SUBAPPLICATION Select_EnableOk (* Leitet aus 2 Bools (bEnable + bOk) einen von 3 Werten ab: valDisabled (bEnable=FALSE) / valOk (bEnable=TRUE, bOk=TRUE) / valFault (bEnable=TRUE, bOk=FALSE). Generischer 2-stufiger F_SEL - die 3 Werte sind Parameter, nicht auf Farben beschraenkt. *)
  (* Standard: 61499-2; Description: Copyright (c) 2026 Meisterschulen am Ostbahnhof This program and the accompanying materials are made available under the terms of the Eclipse Public License 2.0 which is available at https://www.eclipse.org/legal/epl-2.0/ SPDX-License-Identifier: EPL-2.0 *)
  (* Version 1.0, 2026-08-31, Franz Höpfinger, Meisterschulen am Ostbahnhof, Extrahiert aus Q_BackgroundColour_EnableOk - die reine 2-Bool-zu-1-von-3-Werten-Logik, entkoppelt von der VT-Hintergrundfarben-Anwendung *)
  PACKAGE MyLib::sys;
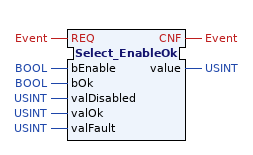
  EVENT_INPUT
    REQ; (* Neu auswerten - bEnable und bOk werden zusammen mitgegeben *)
  END_EVENT
  EVENT_OUTPUT
    CNF; (* Wert berechnet *)
  END_EVENT
  VAR_INPUT
    bEnable : BOOL; (* Aktiviert *)
    bOk : BOOL; (* OK-Zustand (nur relevant wenn bEnable=TRUE) *)
    valDisabled : USINT; (* Ausgabewert wenn bEnable=FALSE - einmalig bei Instanziierung per Parameter gesetzt *)
    valOk : USINT; (* Ausgabewert wenn bEnable=TRUE und bOk=TRUE - einmalig bei Instanziierung per Parameter gesetzt *)
    valFault : USINT; (* Ausgabewert wenn bEnable=TRUE und bOk=FALSE - einmalig bei Instanziierung per Parameter gesetzt *)
  END_VAR
  VAR_OUTPUT
    value : USINT; (* Ausgewaehlter Wert *)
  END_VAR
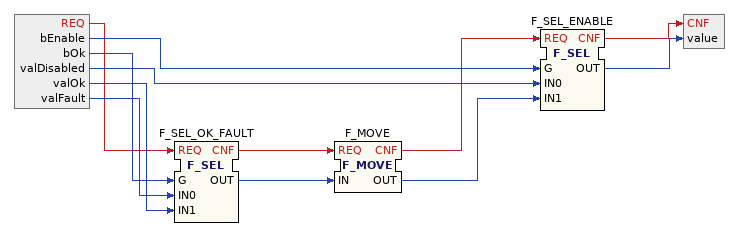
  FBS
    F_SEL_OK_FAULT : iec61131::selection::F_SEL;
    F_MOVE : iec61131::selection::F_MOVE; {SET_ATTRIBUTE(DataType, USINT)}
    F_SEL_ENABLE : iec61131::selection::F_SEL;
  END_FBS
  EVENT_CONNECTIONS
    REQ TO F_SEL_OK_FAULT.REQ;
    F_SEL_OK_FAULT.CNF TO F_MOVE.REQ;
    F_MOVE.CNF TO F_SEL_ENABLE.REQ;
    F_SEL_ENABLE.CNF TO CNF;
  END_CONNECTIONS
  DATA_CONNECTIONS
    bOk TO F_SEL_OK_FAULT.G;
    valFault TO F_SEL_OK_FAULT.IN0;
    valOk TO F_SEL_OK_FAULT.IN1;
    F_SEL_OK_FAULT.OUT TO F_MOVE.IN;
    bEnable TO F_SEL_ENABLE.G;
    valDisabled TO F_SEL_ENABLE.IN0;
    F_MOVE.OUT TO F_SEL_ENABLE.IN1;
    F_SEL_ENABLE.OUT TO value;
  END_CONNECTIONS
END_SUBAPPLICATION
